TYPE Regelungsmethode :
(
	Kraftkreis,
	On_Off
	
	
);
END_TYPE

(* stored: Version 1.1.0.1, ProductVersion 3.1.4024.11
   DUT Regelungsmethode: Id {0c0d245a-f223-42a3-8e5a-7bae4dd90cd0} *)
